TYPE E_SetupPlantStateShape :
(
	eSetupPlantStateShape_None := 0,
	eSetupPlantStateShape_Nok,
	eSetupPlantStateShape_Ok,
	
	
	eSetupPlantStateShape_Max
);
END_TYPE

(* stored: Version 1.1.0.1, ProductVersion 3.1.4024.4
   DUT E_SetupPlantStateShape: Id {19086cd9-40d4-493b-b8fa-a4d445b0086e} *)
